{attribute addProperty BoxType "APS1003-5000-0016"}
{attribute addProperty Id "StatusAT %I*LWORD6481A0_X_FieldAT %I*INT1621A0_Y_FieldAT %I*INT1622A0_Z_FieldAT %I*INT1623A2_X_FieldAT %I*INT1624A2_Y_FieldAT %I*INT1625A2_Z_FieldAT %I*INT1626A4_X_FieldAT %I*INT1627A4_Y_FieldAT %I*INT1628A4_Z_FieldAT %I*INT1629A6_X_FieldAT %I*INT16210A6_Y_FieldAT %I*INT16211A6_Z_FieldAT %I*INT16212A8_X_FieldAT %I*INT16213A8_Y_FieldAT %I*INT16214A8_Z_FieldAT %I*INT16215B1_X_FieldAT %I*INT1621B1_Y_FieldAT %I*INT1622B1_Z_FieldAT %I*INT1623B3_X_FieldAT %I*INT1624B3_Y_FieldAT %I*INT1625B3_Z_FieldAT %I*INT1626B5_X_FieldAT %I*INT1627B5_Y_FieldAT %I*INT1628B5_Z_FieldAT %I*INT1629B7_X_FieldAT %I*INT16210B7_Y_FieldAT %I*INT16211B7_Z_FieldAT %I*INT16212B9_X_FieldAT %I*INT16213B9_Y_FieldAT %I*INT16214B9_Z_FieldAT %I*INT16215C0_X_FieldAT %I*INT1621C0_Y_FieldAT %I*INT1622C0_Z_FieldAT %I*INT1623C2_X_FieldAT %I*INT1624C2_Y_FieldAT %I*INT1625C2_Z_FieldAT %I*INT1626C4_X_FieldAT %I*INT1627C4_Y_FieldAT %I*INT1628C4_Z_FieldAT %I*INT1629C6_X_FieldAT %I*INT16210C6_Y_FieldAT %I*INT16211C6_Z_FieldAT %I*INT16212C8_X_FieldAT %I*INT16213C8_Y_FieldAT %I*INT16214C8_Z_FieldAT %I*INT16215D1_X_FieldAT %I*INT1621D1_Y_FieldAT %I*INT1622D1_Z_FieldAT %I*INT1623D3_X_FieldAT %I*INT1624D3_Y_FieldAT %I*INT1625D3_Z_FieldAT %I*INT1626D5_X_FieldAT %I*INT1627D5_Y_FieldAT %I*INT1628D5_Z_FieldAT %I*INT1629D7_X_FieldAT %I*INT16210D7_Y_FieldAT %I*INT16211D7_Z_FieldAT %I*INT16212D9_X_FieldAT %I*INT16213D9_Y_FieldAT %I*INT16214D9_Z_FieldAT %I*INT16215E0_X_FieldAT %I*INT1621E0_Y_FieldAT %I*INT1622E0_Z_FieldAT %I*INT1623E2_X_FieldAT %I*INT1624E2_Y_FieldAT %I*INT1625E2_Z_FieldAT %I*INT1626E4_X_FieldAT %I*INT1627E4_Y_FieldAT %I*INT1628E4_Z_FieldAT %I*INT1629E6_X_FieldAT %I*INT16210E6_Y_FieldAT %I*INT16211E6_Z_FieldAT %I*INT16212E8_X_FieldAT %I*INT16213E8_Y_FieldAT %I*INT16214E8_Z_FieldAT %I*INT16215F1_X_FieldAT %I*INT1621F1_Y_FieldAT %I*INT1622F1_Z_FieldAT %I*INT1623F3_X_FieldAT %I*INT1624F3_Y_FieldAT %I*INT1625F3_Z_FieldAT %I*INT1626F5_X_FieldAT %I*INT1627F5_Y_FieldAT %I*INT1628F5_Z_FieldAT %I*INT1629F7_X_FieldAT %I*INT16210F7_Y_FieldAT %I*INT16211F7_Z_FieldAT %I*INT16212F9_X_FieldAT %I*INT16213F9_Y_FieldAT %I*INT16214F9_Z_FieldAT %I*INT16215G0_X_FieldAT %I*INT1621G0_Y_FieldAT %I*INT1622G0_Z_FieldAT %I*INT1623G2_X_FieldAT %I*INT1624G2_Y_FieldAT %I*INT1625G2_Z_FieldAT %I*INT1626G4_X_FieldAT %I*INT1627G4_Y_FieldAT %I*INT1628G4_Z_FieldAT %I*INT1629G6_X_FieldAT %I*INT16210G6_Y_FieldAT %I*INT16211G6_Z_FieldAT %I*INT16212G8_X_FieldAT %I*INT16213G8_Y_FieldAT %I*INT16214G8_Z_FieldAT %I*INT16215H1_X_FieldAT %I*INT1621H1_Y_FieldAT %I*INT1622H1_Z_FieldAT %I*INT1623H3_X_FieldAT %I*INT1624H3_Y_FieldAT %I*INT1625H3_Z_FieldAT %I*INT1626H5_X_FieldAT %I*INT1627H5_Y_FieldAT %I*INT1628H5_Z_FieldAT %I*INT1629H7_X_FieldAT %I*INT16210H7_Y_FieldAT %I*INT16211H7_Z_FieldAT %I*INT16212H9_X_FieldAT %I*INT16213H9_Y_FieldAT %I*INT16214H9_Z_FieldAT %I*INT16215I0_X_FieldAT %I*INT1621I0_Y_FieldAT %I*INT1622I0_Z_FieldAT %I*INT1623I2_X_FieldAT %I*INT1624I2_Y_FieldAT %I*INT1625I2_Z_FieldAT %I*INT1626I4_X_FieldAT %I*INT1627I4_Y_FieldAT %I*INT1628I4_Z_FieldAT %I*INT1629I6_X_FieldAT %I*INT16210I6_Y_FieldAT %I*INT16211I6_Z_FieldAT %I*INT16212I8_X_FieldAT %I*INT16213I8_Y_FieldAT %I*INT16214I8_Z_FieldAT %I*INT16215J1_X_FieldAT %I*INT1621J1_Y_FieldAT %I*INT1622J1_Z_FieldAT %I*INT1623J3_X_FieldAT %I*INT1624J3_Y_FieldAT %I*INT1625J3_Z_FieldAT %I*INT1626J5_X_FieldAT %I*INT1627J5_Y_FieldAT %I*INT1628J5_Z_FieldAT %I*INT1629J7_X_FieldAT %I*INT16210J7_Y_FieldAT %I*INT16211J7_Z_FieldAT %I*INT16212J9_X_FieldAT %I*INT16213J9_Y_FieldAT %I*INT16214J9_Z_FieldAT %I*INT16215"}
{attribute addProperty CRC "610062764"}
{attribute addProperty SizeInBites "2464"}
{attribute addProperty SizeInBytes "308"}
TYPE FB_Inputs_245CD1AC :
STRUCT
	{attribute addProperty Name "Status"}
	Status AT %I* : LWORD;
	{attribute addProperty Name "A0_X_Field"}
	A0_X_Field AT %I* : INT;
	{attribute addProperty Name "A0_Y_Field"}
	A0_Y_Field AT %I* : INT;
	{attribute addProperty Name "A0_Z_Field"}
	A0_Z_Field AT %I* : INT;
	{attribute addProperty Name "A2_X_Field"}
	A2_X_Field AT %I* : INT;
	{attribute addProperty Name "A2_Y_Field"}
	A2_Y_Field AT %I* : INT;
	{attribute addProperty Name "A2_Z_Field"}
	A2_Z_Field AT %I* : INT;
	{attribute addProperty Name "A4_X_Field"}
	A4_X_Field AT %I* : INT;
	{attribute addProperty Name "A4_Y_Field"}
	A4_Y_Field AT %I* : INT;
	{attribute addProperty Name "A4_Z_Field"}
	A4_Z_Field AT %I* : INT;
	{attribute addProperty Name "A6_X_Field"}
	A6_X_Field AT %I* : INT;
	{attribute addProperty Name "A6_Y_Field"}
	A6_Y_Field AT %I* : INT;
	{attribute addProperty Name "A6_Z_Field"}
	A6_Z_Field AT %I* : INT;
	{attribute addProperty Name "A8_X_Field"}
	A8_X_Field AT %I* : INT;
	{attribute addProperty Name "A8_Y_Field"}
	A8_Y_Field AT %I* : INT;
	{attribute addProperty Name "A8_Z_Field"}
	A8_Z_Field AT %I* : INT;
	{attribute addProperty Name "B1_X_Field"}
	B1_X_Field AT %I* : INT;
	{attribute addProperty Name "B1_Y_Field"}
	B1_Y_Field AT %I* : INT;
	{attribute addProperty Name "B1_Z_Field"}
	B1_Z_Field AT %I* : INT;
	{attribute addProperty Name "B3_X_Field"}
	B3_X_Field AT %I* : INT;
	{attribute addProperty Name "B3_Y_Field"}
	B3_Y_Field AT %I* : INT;
	{attribute addProperty Name "B3_Z_Field"}
	B3_Z_Field AT %I* : INT;
	{attribute addProperty Name "B5_X_Field"}
	B5_X_Field AT %I* : INT;
	{attribute addProperty Name "B5_Y_Field"}
	B5_Y_Field AT %I* : INT;
	{attribute addProperty Name "B5_Z_Field"}
	B5_Z_Field AT %I* : INT;
	{attribute addProperty Name "B7_X_Field"}
	B7_X_Field AT %I* : INT;
	{attribute addProperty Name "B7_Y_Field"}
	B7_Y_Field AT %I* : INT;
	{attribute addProperty Name "B7_Z_Field"}
	B7_Z_Field AT %I* : INT;
	{attribute addProperty Name "B9_X_Field"}
	B9_X_Field AT %I* : INT;
	{attribute addProperty Name "B9_Y_Field"}
	B9_Y_Field AT %I* : INT;
	{attribute addProperty Name "B9_Z_Field"}
	B9_Z_Field AT %I* : INT;
	{attribute addProperty Name "C0_X_Field"}
	C0_X_Field AT %I* : INT;
	{attribute addProperty Name "C0_Y_Field"}
	C0_Y_Field AT %I* : INT;
	{attribute addProperty Name "C0_Z_Field"}
	C0_Z_Field AT %I* : INT;
	{attribute addProperty Name "C2_X_Field"}
	C2_X_Field AT %I* : INT;
	{attribute addProperty Name "C2_Y_Field"}
	C2_Y_Field AT %I* : INT;
	{attribute addProperty Name "C2_Z_Field"}
	C2_Z_Field AT %I* : INT;
	{attribute addProperty Name "C4_X_Field"}
	C4_X_Field AT %I* : INT;
	{attribute addProperty Name "C4_Y_Field"}
	C4_Y_Field AT %I* : INT;
	{attribute addProperty Name "C4_Z_Field"}
	C4_Z_Field AT %I* : INT;
	{attribute addProperty Name "C6_X_Field"}
	C6_X_Field AT %I* : INT;
	{attribute addProperty Name "C6_Y_Field"}
	C6_Y_Field AT %I* : INT;
	{attribute addProperty Name "C6_Z_Field"}
	C6_Z_Field AT %I* : INT;
	{attribute addProperty Name "C8_X_Field"}
	C8_X_Field AT %I* : INT;
	{attribute addProperty Name "C8_Y_Field"}
	C8_Y_Field AT %I* : INT;
	{attribute addProperty Name "C8_Z_Field"}
	C8_Z_Field AT %I* : INT;
	{attribute addProperty Name "D1_X_Field"}
	D1_X_Field AT %I* : INT;
	{attribute addProperty Name "D1_Y_Field"}
	D1_Y_Field AT %I* : INT;
	{attribute addProperty Name "D1_Z_Field"}
	D1_Z_Field AT %I* : INT;
	{attribute addProperty Name "D3_X_Field"}
	D3_X_Field AT %I* : INT;
	{attribute addProperty Name "D3_Y_Field"}
	D3_Y_Field AT %I* : INT;
	{attribute addProperty Name "D3_Z_Field"}
	D3_Z_Field AT %I* : INT;
	{attribute addProperty Name "D5_X_Field"}
	D5_X_Field AT %I* : INT;
	{attribute addProperty Name "D5_Y_Field"}
	D5_Y_Field AT %I* : INT;
	{attribute addProperty Name "D5_Z_Field"}
	D5_Z_Field AT %I* : INT;
	{attribute addProperty Name "D7_X_Field"}
	D7_X_Field AT %I* : INT;
	{attribute addProperty Name "D7_Y_Field"}
	D7_Y_Field AT %I* : INT;
	{attribute addProperty Name "D7_Z_Field"}
	D7_Z_Field AT %I* : INT;
	{attribute addProperty Name "D9_X_Field"}
	D9_X_Field AT %I* : INT;
	{attribute addProperty Name "D9_Y_Field"}
	D9_Y_Field AT %I* : INT;
	{attribute addProperty Name "D9_Z_Field"}
	D9_Z_Field AT %I* : INT;
	{attribute addProperty Name "E0_X_Field"}
	E0_X_Field AT %I* : INT;
	{attribute addProperty Name "E0_Y_Field"}
	E0_Y_Field AT %I* : INT;
	{attribute addProperty Name "E0_Z_Field"}
	E0_Z_Field AT %I* : INT;
	{attribute addProperty Name "E2_X_Field"}
	E2_X_Field AT %I* : INT;
	{attribute addProperty Name "E2_Y_Field"}
	E2_Y_Field AT %I* : INT;
	{attribute addProperty Name "E2_Z_Field"}
	E2_Z_Field AT %I* : INT;
	{attribute addProperty Name "E4_X_Field"}
	E4_X_Field AT %I* : INT;
	{attribute addProperty Name "E4_Y_Field"}
	E4_Y_Field AT %I* : INT;
	{attribute addProperty Name "E4_Z_Field"}
	E4_Z_Field AT %I* : INT;
	{attribute addProperty Name "E6_X_Field"}
	E6_X_Field AT %I* : INT;
	{attribute addProperty Name "E6_Y_Field"}
	E6_Y_Field AT %I* : INT;
	{attribute addProperty Name "E6_Z_Field"}
	E6_Z_Field AT %I* : INT;
	{attribute addProperty Name "E8_X_Field"}
	E8_X_Field AT %I* : INT;
	{attribute addProperty Name "E8_Y_Field"}
	E8_Y_Field AT %I* : INT;
	{attribute addProperty Name "E8_Z_Field"}
	E8_Z_Field AT %I* : INT;
	{attribute addProperty Name "F1_X_Field"}
	F1_X_Field AT %I* : INT;
	{attribute addProperty Name "F1_Y_Field"}
	F1_Y_Field AT %I* : INT;
	{attribute addProperty Name "F1_Z_Field"}
	F1_Z_Field AT %I* : INT;
	{attribute addProperty Name "F3_X_Field"}
	F3_X_Field AT %I* : INT;
	{attribute addProperty Name "F3_Y_Field"}
	F3_Y_Field AT %I* : INT;
	{attribute addProperty Name "F3_Z_Field"}
	F3_Z_Field AT %I* : INT;
	{attribute addProperty Name "F5_X_Field"}
	F5_X_Field AT %I* : INT;
	{attribute addProperty Name "F5_Y_Field"}
	F5_Y_Field AT %I* : INT;
	{attribute addProperty Name "F5_Z_Field"}
	F5_Z_Field AT %I* : INT;
	{attribute addProperty Name "F7_X_Field"}
	F7_X_Field AT %I* : INT;
	{attribute addProperty Name "F7_Y_Field"}
	F7_Y_Field AT %I* : INT;
	{attribute addProperty Name "F7_Z_Field"}
	F7_Z_Field AT %I* : INT;
	{attribute addProperty Name "F9_X_Field"}
	F9_X_Field AT %I* : INT;
	{attribute addProperty Name "F9_Y_Field"}
	F9_Y_Field AT %I* : INT;
	{attribute addProperty Name "F9_Z_Field"}
	F9_Z_Field AT %I* : INT;
	{attribute addProperty Name "G0_X_Field"}
	G0_X_Field AT %I* : INT;
	{attribute addProperty Name "G0_Y_Field"}
	G0_Y_Field AT %I* : INT;
	{attribute addProperty Name "G0_Z_Field"}
	G0_Z_Field AT %I* : INT;
	{attribute addProperty Name "G2_X_Field"}
	G2_X_Field AT %I* : INT;
	{attribute addProperty Name "G2_Y_Field"}
	G2_Y_Field AT %I* : INT;
	{attribute addProperty Name "G2_Z_Field"}
	G2_Z_Field AT %I* : INT;
	{attribute addProperty Name "G4_X_Field"}
	G4_X_Field AT %I* : INT;
	{attribute addProperty Name "G4_Y_Field"}
	G4_Y_Field AT %I* : INT;
	{attribute addProperty Name "G4_Z_Field"}
	G4_Z_Field AT %I* : INT;
	{attribute addProperty Name "G6_X_Field"}
	G6_X_Field AT %I* : INT;
	{attribute addProperty Name "G6_Y_Field"}
	G6_Y_Field AT %I* : INT;
	{attribute addProperty Name "G6_Z_Field"}
	G6_Z_Field AT %I* : INT;
	{attribute addProperty Name "G8_X_Field"}
	G8_X_Field AT %I* : INT;
	{attribute addProperty Name "G8_Y_Field"}
	G8_Y_Field AT %I* : INT;
	{attribute addProperty Name "G8_Z_Field"}
	G8_Z_Field AT %I* : INT;
	{attribute addProperty Name "H1_X_Field"}
	H1_X_Field AT %I* : INT;
	{attribute addProperty Name "H1_Y_Field"}
	H1_Y_Field AT %I* : INT;
	{attribute addProperty Name "H1_Z_Field"}
	H1_Z_Field AT %I* : INT;
	{attribute addProperty Name "H3_X_Field"}
	H3_X_Field AT %I* : INT;
	{attribute addProperty Name "H3_Y_Field"}
	H3_Y_Field AT %I* : INT;
	{attribute addProperty Name "H3_Z_Field"}
	H3_Z_Field AT %I* : INT;
	{attribute addProperty Name "H5_X_Field"}
	H5_X_Field AT %I* : INT;
	{attribute addProperty Name "H5_Y_Field"}
	H5_Y_Field AT %I* : INT;
	{attribute addProperty Name "H5_Z_Field"}
	H5_Z_Field AT %I* : INT;
	{attribute addProperty Name "H7_X_Field"}
	H7_X_Field AT %I* : INT;
	{attribute addProperty Name "H7_Y_Field"}
	H7_Y_Field AT %I* : INT;
	{attribute addProperty Name "H7_Z_Field"}
	H7_Z_Field AT %I* : INT;
	{attribute addProperty Name "H9_X_Field"}
	H9_X_Field AT %I* : INT;
	{attribute addProperty Name "H9_Y_Field"}
	H9_Y_Field AT %I* : INT;
	{attribute addProperty Name "H9_Z_Field"}
	H9_Z_Field AT %I* : INT;
	{attribute addProperty Name "I0_X_Field"}
	I0_X_Field AT %I* : INT;
	{attribute addProperty Name "I0_Y_Field"}
	I0_Y_Field AT %I* : INT;
	{attribute addProperty Name "I0_Z_Field"}
	I0_Z_Field AT %I* : INT;
	{attribute addProperty Name "I2_X_Field"}
	I2_X_Field AT %I* : INT;
	{attribute addProperty Name "I2_Y_Field"}
	I2_Y_Field AT %I* : INT;
	{attribute addProperty Name "I2_Z_Field"}
	I2_Z_Field AT %I* : INT;
	{attribute addProperty Name "I4_X_Field"}
	I4_X_Field AT %I* : INT;
	{attribute addProperty Name "I4_Y_Field"}
	I4_Y_Field AT %I* : INT;
	{attribute addProperty Name "I4_Z_Field"}
	I4_Z_Field AT %I* : INT;
	{attribute addProperty Name "I6_X_Field"}
	I6_X_Field AT %I* : INT;
	{attribute addProperty Name "I6_Y_Field"}
	I6_Y_Field AT %I* : INT;
	{attribute addProperty Name "I6_Z_Field"}
	I6_Z_Field AT %I* : INT;
	{attribute addProperty Name "I8_X_Field"}
	I8_X_Field AT %I* : INT;
	{attribute addProperty Name "I8_Y_Field"}
	I8_Y_Field AT %I* : INT;
	{attribute addProperty Name "I8_Z_Field"}
	I8_Z_Field AT %I* : INT;
	{attribute addProperty Name "J1_X_Field"}
	J1_X_Field AT %I* : INT;
	{attribute addProperty Name "J1_Y_Field"}
	J1_Y_Field AT %I* : INT;
	{attribute addProperty Name "J1_Z_Field"}
	J1_Z_Field AT %I* : INT;
	{attribute addProperty Name "J3_X_Field"}
	J3_X_Field AT %I* : INT;
	{attribute addProperty Name "J3_Y_Field"}
	J3_Y_Field AT %I* : INT;
	{attribute addProperty Name "J3_Z_Field"}
	J3_Z_Field AT %I* : INT;
	{attribute addProperty Name "J5_X_Field"}
	J5_X_Field AT %I* : INT;
	{attribute addProperty Name "J5_Y_Field"}
	J5_Y_Field AT %I* : INT;
	{attribute addProperty Name "J5_Z_Field"}
	J5_Z_Field AT %I* : INT;
	{attribute addProperty Name "J7_X_Field"}
	J7_X_Field AT %I* : INT;
	{attribute addProperty Name "J7_Y_Field"}
	J7_Y_Field AT %I* : INT;
	{attribute addProperty Name "J7_Z_Field"}
	J7_Z_Field AT %I* : INT;
	{attribute addProperty Name "J9_X_Field"}
	J9_X_Field AT %I* : INT;
	{attribute addProperty Name "J9_Y_Field"}
	J9_Y_Field AT %I* : INT;
	{attribute addProperty Name "J9_Z_Field"}
	J9_Z_Field AT %I* : INT;
END_STRUCT
END_TYPE

(* stored: Version 1.2.0.0, ProductVersion 3.1.4024.9
   DUT FB_Inputs_245CD1AC: Id {dd82a6f8-e908-480e-8518-e9ae0404eb32} *)
